FUNCTION_BLOCK CmdSludgeDischargeSLBLogic_HMI (* Service Interface Function Block Type *)
  (* Standard: 61499-2 *)
  (* Version 1.0, 10/1/2026, Claude/Hidryco, Schneider Electric, Rev1 - Evento PUMP_STS com o estado das bombas para o simbolo sDefault *)
  PACKAGE SE.Nereda;
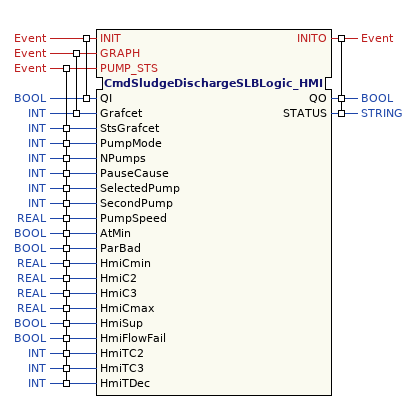
  EVENT_INPUT
    INIT WITH QI;
    GRAPH WITH Grafcet;
    PUMP_STS WITH StsGrafcet, PumpMode, NPumps, PauseCause, SelectedPump, SecondPump, PumpSpeed, AtMin, ParBad, HmiCmin, HmiC2, HmiC3, HmiCmax, HmiSup, HmiFlowFail, HmiTC2, HmiTC3, HmiTDec; (* Status das bombas da descarga *)
  END_EVENT
  EVENT_OUTPUT
    INITO WITH QO, STATUS;
  END_EVENT
  VAR_INPUT
    QI : BOOL;
    Grafcet : INT;
    StsGrafcet : INT;
    PumpMode : INT;
    NPumps : INT;
    PauseCause : INT;
    SelectedPump : INT;
    SecondPump : INT;
    PumpSpeed : REAL;
    AtMin : BOOL;
    ParBad : BOOL;
    HmiCmin : REAL;
    HmiC2 : REAL;
    HmiC3 : REAL;
    HmiCmax : REAL;
    HmiSup : BOOL;
    HmiFlowFail : BOOL;
    HmiTC2 : INT;
    HmiTC3 : INT;
    HmiTDec : INT;
  END_VAR
  VAR_OUTPUT
    QO : BOOL; (* Event Output Qualifier *)
    STATUS : STRING; (* Service Status *)
  END_VAR
  SERVICE /
    SEQUENCE 
    END_SEQUENCE
  END_SERVICE
END_FUNCTION_BLOCK
